// TIA Portal V18 program export: 1 tag tables, 0 data types, 5 data blocks, 11 code blocks (in call order from the OBs), 3 instance data blocks

VAR_GLOBAL   // PLC tag table "Default tag table"
   PB_MAIN_MOVE_R AT %I0.0 : Bool;
   PB_MAIN_MOVE_F AT %I0.1 : Bool;
   PB_MAIN_STOP AT %I0.2 : Bool;
   SENSOR_HOME AT %I0.3 : Bool;
   SENSOR_FINISH_1 AT %I0.4 : Bool;
   PB_EMERGENCY AT %I0.5 : Bool;
   PB_RESET AT %I0.6 : Bool;
   MAIN_COIL_R AT %Q0.0 : Bool;
   MAIN_COIL_F AT %Q0.1 : Bool;
   COIL_EMERGENCY AT %Q0.2 : Bool;
   System_Byte AT %MB1 : Byte;
   FirstScan AT %M1.0 : Bool;
   DiagStatusUpdate AT %M1.1 : Bool;
   AlwaysTRUE AT %M1.2 : Bool;
   AlwaysFALSE AT %M1.3 : Bool;
   Clock_Byte AT %MB0 : Byte;
   Clock_10Hz AT %M0.0 : Bool;
   Clock_5Hz AT %M0.1 : Bool;
   "Clock_2.5Hz" AT %M0.2 : Bool;
   Clock_2Hz AT %M0.3 : Bool;
   "Clock_1.25Hz" AT %M0.4 : Bool;
   Clock_1Hz AT %M0.5 : Bool;
   "Clock_0.625Hz" AT %M0.6 : Bool;
   "Clock_0.5Hz" AT %M0.7 : Bool;
   M1_RESET_COUNT AT %I0.7 : Bool;
   PB_M1_MOVE_R AT %I1.0 : Bool;
   PB_M1_MOVE_F AT %I1.1 : Bool;
   PB_M1_STOP AT %I1.2 : Bool;
   M1_COIL_R AT %Q0.3 : Bool;
   M1_COIL_F AT %Q0.4 : Bool;
   SENSOR_FINISH_2 AT %I1.3 : Bool;
   M2_RESET_COUNTER AT %I1.4 : Bool;
   PB_M2_MOVE_R AT %I1.5 : Bool;
   M2_COIL_R AT %Q0.5 : Bool;
   M2_COIL_F AT %Q0.6 : Bool;
   PB_M2_MOVE_F AT %I8.0 : Bool;
   PB_M2_STOP AT %I8.1 : Bool;
   DIVIDER_1 AT %Q8.0 : Bool;
   DIVIDER_2 AT %Q8.1 : Bool;
END_VAR

DATA_BLOCK "HMI_DB"   // DB20
{ S7_Optimized_Access := 'FALSE' }
VERSION : 0.1
// stored: AutoNumber true, DBAccessibleFromOPCUA true, IsOnlyStoredInLoadMemory false, IsWriteProtectedInAS false
   VAR
      MAIN_MOVE_F : Bool;
      MAIN_MOVE_R : Bool;
      MAIN_STOP : Bool;
      EMERGENCY : Bool;
      RESET : Bool;
      M1_MOVE_F : Bool;
      M1_MOVE_R : Bool;
      M1_STOP : Bool;
      RESET_COUNTER_1 : Bool;
      M2_MOVE_F : Bool;
      M2_MOVE_R : Bool;
      M2_STOP : Bool;
      RESET_COUNTER_2 : Bool;
      MAIN_FORWARD : Bool;
      MAIN_REVERSE : Bool;
      M1_FORWARD : Bool;
      M1_REVERSE : Bool;
      M2_FORWARD : Bool;
      M2_REVERSE : Bool;
   END_VAR
BEGIN
END_DATA_BLOCK

DATA_BLOCK "M1_I/O_DB"   // DB7
{ S7_Optimized_Access := 'FALSE' }
VERSION : 0.1
// stored: AutoNumber true, DBAccessibleFromOPCUA true, IsOnlyStoredInLoadMemory false, IsWriteProtectedInAS false
   VAR
      RESET_COUNTER : Bool;
      M1_MOVE_R : Bool;
      M1_MOVE_F : Bool;
      M1_STOP : Bool;
   END_VAR
BEGIN
END_DATA_BLOCK

DATA_BLOCK "M2_I/O_DB"   // DB19
{ S7_Optimized_Access := 'FALSE' }
VERSION : 0.1
// stored: AutoNumber true, DBAccessibleFromOPCUA true, IsOnlyStoredInLoadMemory false, IsWriteProtectedInAS false
   VAR
      RESET_COUNTER : Bool;
      M2_MOVE_R : Bool;
      M2_MOVE_F : Bool;
      M2_STOP : Bool;
   END_VAR
BEGIN
END_DATA_BLOCK

DATA_BLOCK "MAIN_I/O_DB"   // DB1
{ S7_Optimized_Access := 'FALSE' }
VERSION : 0.1
// stored: AutoNumber true, DBAccessibleFromOPCUA true, IsOnlyStoredInLoadMemory false, IsWriteProtectedInAS false
   VAR
      MAIN_MOVE_R : Bool;
      MAIN_MOVE_F : Bool;
      MAIN_STOP : Bool;
      SENSOR_HOME : Bool;
      SENSOR_FINISH_1 : Bool;
      SENSOR_FINISH_2 : Bool;
      EMERGENCY : Bool;
      RESET : Bool;
      MAIN_COIL_F : Bool;
      MAIN_COIL_R : Bool;
      COIL_EMERGENCY : Bool;
   END_VAR
BEGIN
END_DATA_BLOCK

DATA_BLOCK "STATES_DB"   // DB2
{ S7_Optimized_Access := 'FALSE' }
VERSION : 0.1
// stored: AutoNumber true, DBAccessibleFromOPCUA true, IsOnlyStoredInLoadMemory false, IsWriteProtectedInAS false
   VAR
      EMERGENCY_STATE : Bool;
      DIV_1 : Bool;
      DIV_2 : Bool;
      MAIN_WIND_DOWN : Bool;
      M1_WIND_DOWN : Bool;
      M2_WIND_DOWN : Bool;
      DIV1_COUNTING_READY : Bool;
      DIV2_COUNTING_READY : Bool;
   END_VAR
BEGIN
END_DATA_BLOCK

ORGANIZATION_BLOCK "Main"   // OB1, LAD, ProgramCycle
TITLE = "Main Program Sweep (Cycle)"
{ S7_Optimized_Access := 'TRUE' }
VERSION : 0.1
// stored: AutoNumber true, IsIECCheckEnabled false, SetENOAutomatically false
   VAR_INPUT
      Initial_Call : Bool;   // Initial call of this OB
      Remanence : Bool;   // =True, if remanent data are available
   END_VAR
BEGIN

REGION Network 1
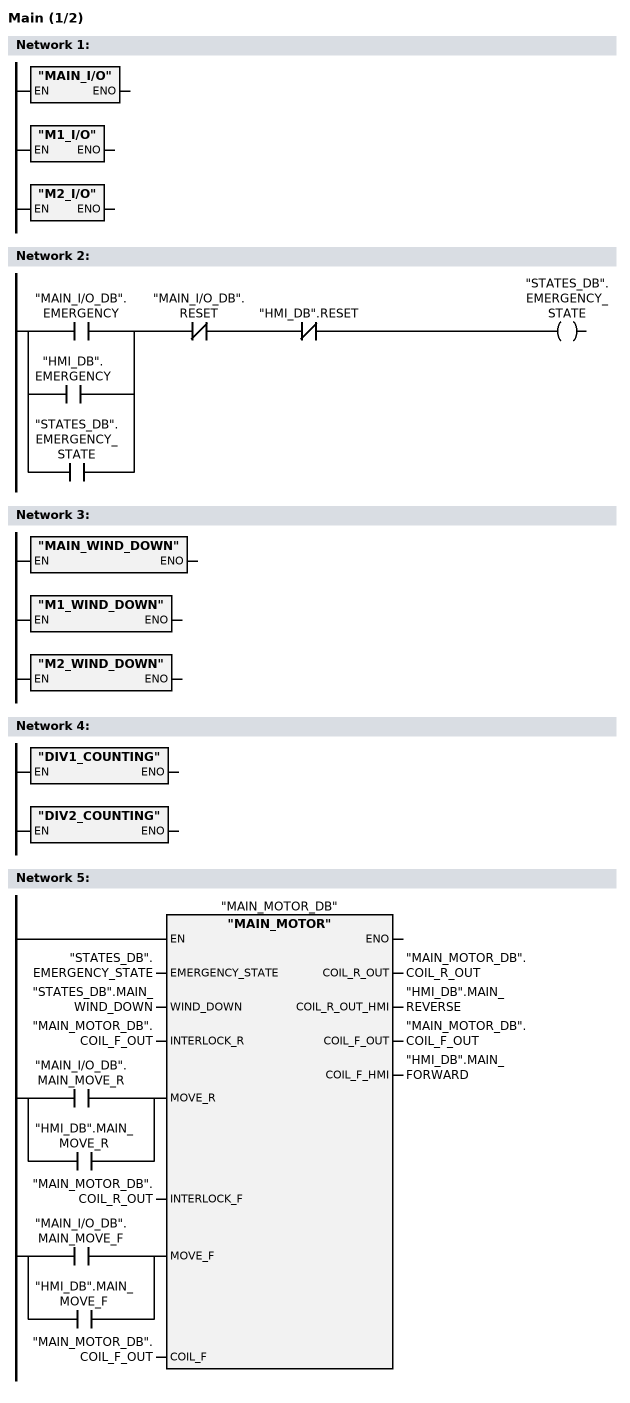
   RUNG wire#powerrail
      "MAIN_I/O"()
   END_RUNG
   RUNG wire#powerrail
      "M1_I/O"()
   END_RUNG
   RUNG wire#powerrail
      "M2_I/O"()
   END_RUNG
   // the same network as SCL:
   "MAIN_I/O"();
   "M1_I/O"();
   "M2_I/O"();
END_REGION

REGION Network 2
   RUNG wire#powerrail
      Contact( "MAIN_I/O_DB".EMERGENCY )
      wire#w1
      I_Contact( "MAIN_I/O_DB".RESET )
      I_Contact( "HMI_DB".RESET )
      Coil( "STATES_DB".EMERGENCY_STATE )
   END_RUNG
   RUNG wire#powerrail
      Contact( "HMI_DB".EMERGENCY )
   END_RUNG wire#w1
   RUNG wire#powerrail
      Contact( "STATES_DB".EMERGENCY_STATE )
   END_RUNG wire#w1
   // the same network as SCL:
   "STATES_DB".EMERGENCY_STATE := ("MAIN_I/O_DB".EMERGENCY OR "HMI_DB".EMERGENCY OR "STATES_DB".EMERGENCY_STATE) AND NOT "MAIN_I/O_DB".RESET AND NOT "HMI_DB".RESET;
END_REGION

REGION Network 3
   RUNG wire#powerrail
      "MAIN_WIND_DOWN"()
   END_RUNG
   RUNG wire#powerrail
      "M1_WIND_DOWN"()
   END_RUNG
   RUNG wire#powerrail
      "M2_WIND_DOWN"()
   END_RUNG
   // the same network as SCL:
   "MAIN_WIND_DOWN"();
   "M1_WIND_DOWN"();
   "M2_WIND_DOWN"();
END_REGION

REGION Network 4
   RUNG wire#powerrail
      "DIV1_COUNTING"()
   END_RUNG
   RUNG wire#powerrail
      "DIV2_COUNTING"()
   END_RUNG
   // the same network as SCL:
   "DIV1_COUNTING"();
   "DIV2_COUNTING"();
END_REGION

REGION Network 5
   RUNG wire#powerrail
      "MAIN_MOTOR_DB"(MOVE_R := wire#w1, MOVE_F := wire#w2, EMERGENCY_STATE := "STATES_DB".EMERGENCY_STATE, WIND_DOWN := "STATES_DB".MAIN_WIND_DOWN, INTERLOCK_R := "MAIN_MOTOR_DB".COIL_F_OUT, INTERLOCK_F := "MAIN_MOTOR_DB".COIL_R_OUT, COIL_F := "MAIN_MOTOR_DB".COIL_F_OUT, COIL_R_OUT => "MAIN_MOTOR_DB".COIL_R_OUT, COIL_R_OUT_HMI => "HMI_DB".MAIN_REVERSE, COIL_F_OUT => "MAIN_MOTOR_DB".COIL_F_OUT, COIL_F_HMI => "HMI_DB".MAIN_FORWARD)
   END_RUNG
   RUNG wire#powerrail
      Contact( "MAIN_I/O_DB".MAIN_MOVE_R )
   END_RUNG wire#w1
   RUNG wire#powerrail
      Contact( "HMI_DB".MAIN_MOVE_R )
   END_RUNG wire#w1
   RUNG wire#powerrail
      Contact( "MAIN_I/O_DB".MAIN_MOVE_F )
   END_RUNG wire#w2
   RUNG wire#powerrail
      Contact( "HMI_DB".MAIN_MOVE_F )
   END_RUNG wire#w2
   // the same network as SCL:
   "MAIN_MOTOR_DB"(EMERGENCY_STATE := "STATES_DB".EMERGENCY_STATE,   // "MAIN_MOTOR"
                   WIND_DOWN := "STATES_DB".MAIN_WIND_DOWN,
                   INTERLOCK_R := "MAIN_MOTOR_DB".COIL_F_OUT,
                   MOVE_R := "MAIN_I/O_DB".MAIN_MOVE_R OR "HMI_DB".MAIN_MOVE_R,
                   INTERLOCK_F := "MAIN_MOTOR_DB".COIL_R_OUT,
                   MOVE_F := "MAIN_I/O_DB".MAIN_MOVE_F OR "HMI_DB".MAIN_MOVE_F,
                   COIL_F := "MAIN_MOTOR_DB".COIL_F_OUT,
                   COIL_R_OUT => "MAIN_MOTOR_DB".COIL_R_OUT,
                   COIL_R_OUT_HMI => "HMI_DB".MAIN_REVERSE,
                   COIL_F_OUT => "MAIN_MOTOR_DB".COIL_F_OUT,
                   COIL_F_HMI => "HMI_DB".MAIN_FORWARD);
END_REGION

REGION Network 6
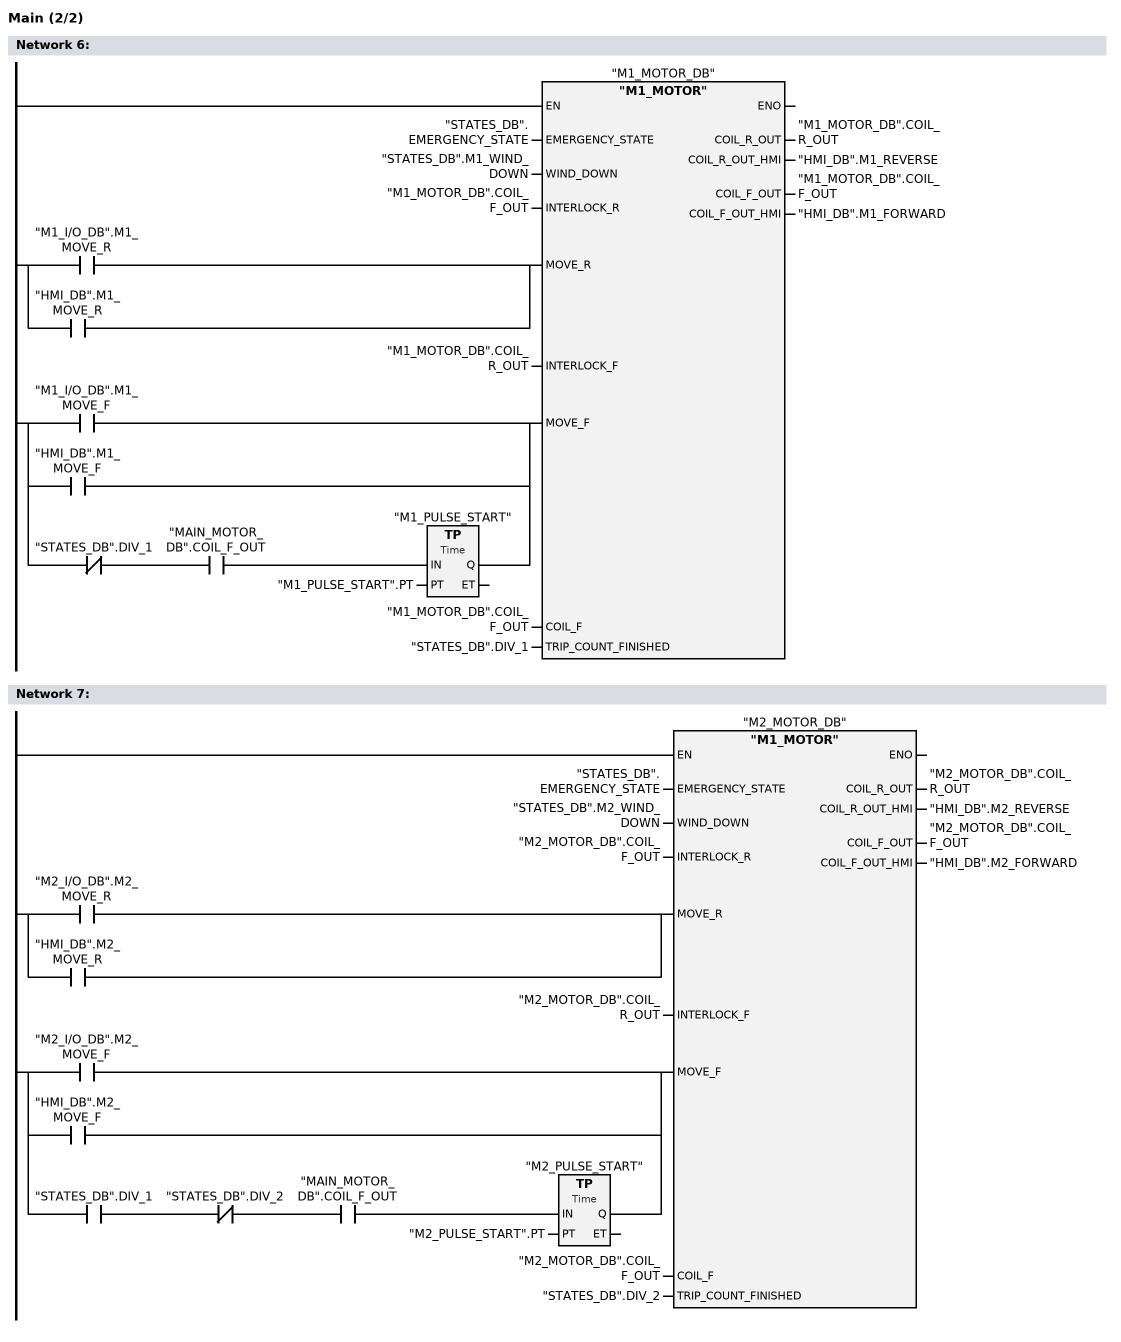
   RUNG wire#powerrail
      "M1_MOTOR_DB"(MOVE_R := wire#w1, MOVE_F := wire#w2, EMERGENCY_STATE := "STATES_DB".EMERGENCY_STATE, WIND_DOWN := "STATES_DB".M1_WIND_DOWN, INTERLOCK_R := "M1_MOTOR_DB".COIL_F_OUT, INTERLOCK_F := "M1_MOTOR_DB".COIL_R_OUT, COIL_F := "M1_MOTOR_DB".COIL_F_OUT, TRIP_COUNT_FINISHED := "STATES_DB".DIV_1, COIL_R_OUT => "M1_MOTOR_DB".COIL_R_OUT, COIL_R_OUT_HMI => "HMI_DB".M1_REVERSE, COIL_F_OUT => "M1_MOTOR_DB".COIL_F_OUT, COIL_F_OUT_HMI => "HMI_DB".M1_FORWARD)
   END_RUNG
   RUNG wire#powerrail
      Contact( "M1_I/O_DB".M1_MOVE_R )
   END_RUNG wire#w1
   RUNG wire#powerrail
      Contact( "HMI_DB".M1_MOVE_R )
   END_RUNG wire#w1
   RUNG wire#powerrail
      Contact( "M1_I/O_DB".M1_MOVE_F )
   END_RUNG wire#w2
   RUNG wire#powerrail
      Contact( "HMI_DB".M1_MOVE_F )
   END_RUNG wire#w2
   RUNG wire#powerrail
      I_Contact( "STATES_DB".DIV_1 )
      Contact( "MAIN_MOTOR_DB".COIL_F_OUT )
      { S7_Templates := "time_type := Time" } "M1_PULSE_START".TP(pt := "M1_PULSE_START".PT, et =>)
   END_RUNG wire#w2
   // the same network as SCL:
   "M1_PULSE_START".TP(IN := NOT "STATES_DB".DIV_1 AND "MAIN_MOTOR_DB".COIL_F_OUT, PT := "M1_PULSE_START".PT);
   "M1_MOTOR_DB"(EMERGENCY_STATE := "STATES_DB".EMERGENCY_STATE,   // "M1_MOTOR"
                 WIND_DOWN := "STATES_DB".M1_WIND_DOWN,
                 INTERLOCK_R := "M1_MOTOR_DB".COIL_F_OUT,
                 MOVE_R := "M1_I/O_DB".M1_MOVE_R OR "HMI_DB".M1_MOVE_R,
                 INTERLOCK_F := "M1_MOTOR_DB".COIL_R_OUT,
                 MOVE_F := "M1_I/O_DB".M1_MOVE_F OR "HMI_DB".M1_MOVE_F OR "M1_PULSE_START".Q,
                 COIL_F := "M1_MOTOR_DB".COIL_F_OUT,
                 TRIP_COUNT_FINISHED := "STATES_DB".DIV_1,
                 COIL_R_OUT => "M1_MOTOR_DB".COIL_R_OUT,
                 COIL_R_OUT_HMI => "HMI_DB".M1_REVERSE,
                 COIL_F_OUT => "M1_MOTOR_DB".COIL_F_OUT,
                 COIL_F_OUT_HMI => "HMI_DB".M1_FORWARD);
END_REGION

REGION Network 7
   RUNG wire#powerrail
      "M2_MOTOR_DB"(MOVE_R := wire#w1, MOVE_F := wire#w2, EMERGENCY_STATE := "STATES_DB".EMERGENCY_STATE, WIND_DOWN := "STATES_DB".M2_WIND_DOWN, INTERLOCK_R := "M2_MOTOR_DB".COIL_F_OUT, INTERLOCK_F := "M2_MOTOR_DB".COIL_R_OUT, COIL_F := "M2_MOTOR_DB".COIL_F_OUT, TRIP_COUNT_FINISHED := "STATES_DB".DIV_2, COIL_R_OUT => "M2_MOTOR_DB".COIL_R_OUT, COIL_R_OUT_HMI => "HMI_DB".M2_REVERSE, COIL_F_OUT => "M2_MOTOR_DB".COIL_F_OUT, COIL_F_OUT_HMI => "HMI_DB".M2_FORWARD)
   END_RUNG
   RUNG wire#powerrail
      Contact( "M2_I/O_DB".M2_MOVE_R )
   END_RUNG wire#w1
   RUNG wire#powerrail
      Contact( "HMI_DB".M2_MOVE_R )
   END_RUNG wire#w1
   RUNG wire#powerrail
      Contact( "M2_I/O_DB".M2_MOVE_F )
   END_RUNG wire#w2
   RUNG wire#powerrail
      Contact( "HMI_DB".M2_MOVE_F )
   END_RUNG wire#w2
   RUNG wire#powerrail
      Contact( "STATES_DB".DIV_1 )
      I_Contact( "STATES_DB".DIV_2 )
      Contact( "MAIN_MOTOR_DB".COIL_F_OUT )
      { S7_Templates := "time_type := Time" } "M2_PULSE_START".TP(pt := "M2_PULSE_START".PT, et =>)
   END_RUNG wire#w2
   // the same network as SCL:
   "M2_PULSE_START".TP(IN := "STATES_DB".DIV_1 AND NOT "STATES_DB".DIV_2 AND "MAIN_MOTOR_DB".COIL_F_OUT,
                       PT := "M2_PULSE_START".PT);
   "M2_MOTOR_DB"(EMERGENCY_STATE := "STATES_DB".EMERGENCY_STATE,   // "M1_MOTOR"
                 WIND_DOWN := "STATES_DB".M2_WIND_DOWN,
                 INTERLOCK_R := "M2_MOTOR_DB".COIL_F_OUT,
                 MOVE_R := "M2_I/O_DB".M2_MOVE_R OR "HMI_DB".M2_MOVE_R,
                 INTERLOCK_F := "M2_MOTOR_DB".COIL_R_OUT,
                 MOVE_F := "M2_I/O_DB".M2_MOVE_F OR "HMI_DB".M2_MOVE_F OR "M2_PULSE_START".Q,
                 COIL_F := "M2_MOTOR_DB".COIL_F_OUT,
                 TRIP_COUNT_FINISHED := "STATES_DB".DIV_2,
                 COIL_R_OUT => "M2_MOTOR_DB".COIL_R_OUT,
                 COIL_R_OUT_HMI => "HMI_DB".M2_REVERSE,
                 COIL_F_OUT => "M2_MOTOR_DB".COIL_F_OUT,
                 COIL_F_OUT_HMI => "HMI_DB".M2_FORWARD);
END_REGION
END_ORGANIZATION_BLOCK

FUNCTION "MAIN_I/O" : Void   // FC1, LAD
{ S7_Optimized_Access := 'TRUE' }
VERSION : 0.1
// stored: AutoNumber true, IsIECCheckEnabled false, SetENOAutomatically false, UDAEnableTagReadback false
BEGIN

REGION Network 1
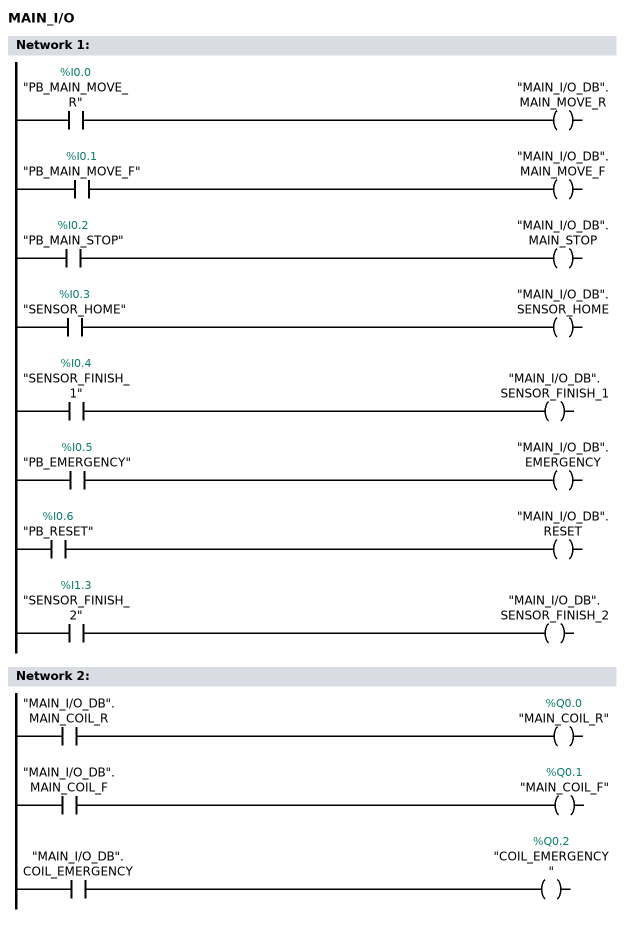
   RUNG wire#powerrail
      Contact( "PB_MAIN_MOVE_R" )
      Coil( "MAIN_I/O_DB".MAIN_MOVE_R )
   END_RUNG
   RUNG wire#powerrail
      Contact( "PB_MAIN_MOVE_F" )
      Coil( "MAIN_I/O_DB".MAIN_MOVE_F )
   END_RUNG
   RUNG wire#powerrail
      Contact( "PB_MAIN_STOP" )
      Coil( "MAIN_I/O_DB".MAIN_STOP )
   END_RUNG
   RUNG wire#powerrail
      Contact( "SENSOR_HOME" )
      Coil( "MAIN_I/O_DB".SENSOR_HOME )
   END_RUNG
   RUNG wire#powerrail
      Contact( "SENSOR_FINISH_1" )
      Coil( "MAIN_I/O_DB".SENSOR_FINISH_1 )
   END_RUNG
   RUNG wire#powerrail
      Contact( "PB_EMERGENCY" )
      Coil( "MAIN_I/O_DB".EMERGENCY )
   END_RUNG
   RUNG wire#powerrail
      Contact( "PB_RESET" )
      Coil( "MAIN_I/O_DB".RESET )
   END_RUNG
   RUNG wire#powerrail
      Contact( "SENSOR_FINISH_2" )
      Coil( "MAIN_I/O_DB".SENSOR_FINISH_2 )
   END_RUNG
   // the same network as SCL:
   "MAIN_I/O_DB".MAIN_MOVE_R := "PB_MAIN_MOVE_R";
   "MAIN_I/O_DB".MAIN_MOVE_F := "PB_MAIN_MOVE_F";
   "MAIN_I/O_DB".MAIN_STOP := "PB_MAIN_STOP";
   "MAIN_I/O_DB".SENSOR_HOME := "SENSOR_HOME";
   "MAIN_I/O_DB".SENSOR_FINISH_1 := "SENSOR_FINISH_1";
   "MAIN_I/O_DB".EMERGENCY := "PB_EMERGENCY";
   "MAIN_I/O_DB".RESET := "PB_RESET";
   "MAIN_I/O_DB".SENSOR_FINISH_2 := "SENSOR_FINISH_2";
END_REGION

REGION Network 2
   RUNG wire#powerrail
      Contact( "MAIN_I/O_DB".MAIN_COIL_R )
      Coil( "MAIN_COIL_R" )
   END_RUNG
   RUNG wire#powerrail
      Contact( "MAIN_I/O_DB".MAIN_COIL_F )
      Coil( "MAIN_COIL_F" )
   END_RUNG
   RUNG wire#powerrail
      Contact( "MAIN_I/O_DB".COIL_EMERGENCY )
      Coil( "COIL_EMERGENCY" )
   END_RUNG
   // the same network as SCL:
   "MAIN_COIL_R" := "MAIN_I/O_DB".MAIN_COIL_R;
   "MAIN_COIL_F" := "MAIN_I/O_DB".MAIN_COIL_F;
   "COIL_EMERGENCY" := "MAIN_I/O_DB".COIL_EMERGENCY;
END_REGION
END_FUNCTION

FUNCTION "M1_I/O" : Void   // FC4, LAD
{ S7_Optimized_Access := 'TRUE' }
VERSION : 0.1
// stored: AutoNumber true, IsIECCheckEnabled false, SetENOAutomatically false, UDAEnableTagReadback false
BEGIN

REGION Network 1
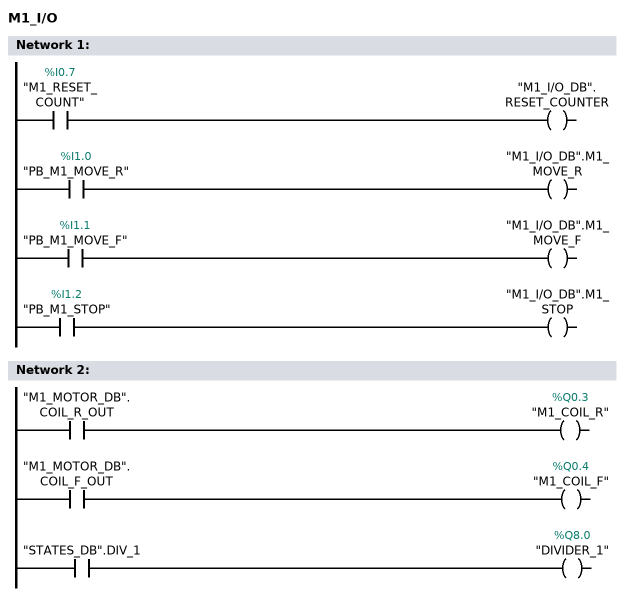
   RUNG wire#powerrail
      Contact( "M1_RESET_COUNT" )
      Coil( "M1_I/O_DB".RESET_COUNTER )
   END_RUNG
   RUNG wire#powerrail
      Contact( "PB_M1_MOVE_R" )
      Coil( "M1_I/O_DB".M1_MOVE_R )
   END_RUNG
   RUNG wire#powerrail
      Contact( "PB_M1_MOVE_F" )
      Coil( "M1_I/O_DB".M1_MOVE_F )
   END_RUNG
   RUNG wire#powerrail
      Contact( "PB_M1_STOP" )
      Coil( "M1_I/O_DB".M1_STOP )
   END_RUNG
   // the same network as SCL:
   "M1_I/O_DB".RESET_COUNTER := "M1_RESET_COUNT";
   "M1_I/O_DB".M1_MOVE_R := "PB_M1_MOVE_R";
   "M1_I/O_DB".M1_MOVE_F := "PB_M1_MOVE_F";
   "M1_I/O_DB".M1_STOP := "PB_M1_STOP";
END_REGION

REGION Network 2
   RUNG wire#powerrail
      Contact( "M1_MOTOR_DB".COIL_R_OUT )
      Coil( "M1_COIL_R" )
   END_RUNG
   RUNG wire#powerrail
      Contact( "M1_MOTOR_DB".COIL_F_OUT )
      Coil( "M1_COIL_F" )
   END_RUNG
   RUNG wire#powerrail
      Contact( "STATES_DB".DIV_1 )
      Coil( "DIVIDER_1" )
   END_RUNG
   // the same network as SCL:
   "M1_COIL_R" := "M1_MOTOR_DB".COIL_R_OUT;
   "M1_COIL_F" := "M1_MOTOR_DB".COIL_F_OUT;
   "DIVIDER_1" := "STATES_DB".DIV_1;
END_REGION
END_FUNCTION

FUNCTION "M2_I/O" : Void   // FC7, LAD
{ S7_Optimized_Access := 'TRUE' }
VERSION : 0.1
// stored: AutoNumber true, IsIECCheckEnabled false, SetENOAutomatically false, UDAEnableTagReadback false
BEGIN

REGION Network 1
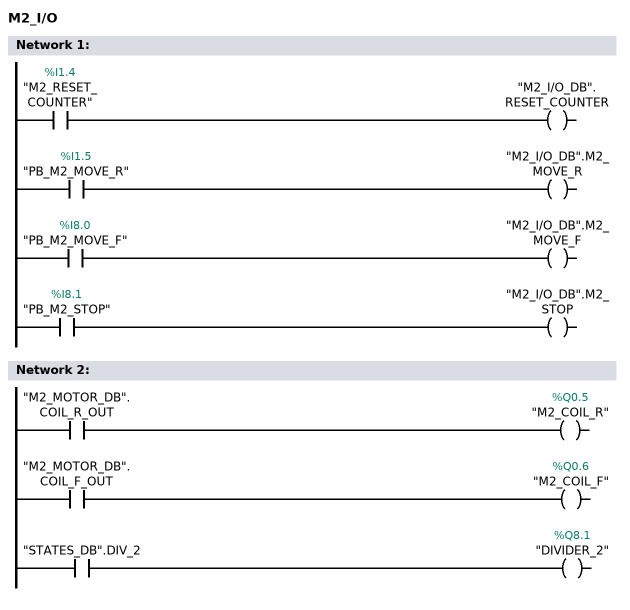
   RUNG wire#powerrail
      Contact( "M2_RESET_COUNTER" )
      Coil( "M2_I/O_DB".RESET_COUNTER )
   END_RUNG
   RUNG wire#powerrail
      Contact( "PB_M2_MOVE_R" )
      Coil( "M2_I/O_DB".M2_MOVE_R )
   END_RUNG
   RUNG wire#powerrail
      Contact( "PB_M2_MOVE_F" )
      Coil( "M2_I/O_DB".M2_MOVE_F )
   END_RUNG
   RUNG wire#powerrail
      Contact( "PB_M2_STOP" )
      Coil( "M2_I/O_DB".M2_STOP )
   END_RUNG
   // the same network as SCL:
   "M2_I/O_DB".RESET_COUNTER := "M2_RESET_COUNTER";
   "M2_I/O_DB".M2_MOVE_R := "PB_M2_MOVE_R";
   "M2_I/O_DB".M2_MOVE_F := "PB_M2_MOVE_F";
   "M2_I/O_DB".M2_STOP := "PB_M2_STOP";
END_REGION

REGION Network 2
   RUNG wire#powerrail
      Contact( "M2_MOTOR_DB".COIL_R_OUT )
      Coil( "M2_COIL_R" )
   END_RUNG
   RUNG wire#powerrail
      Contact( "M2_MOTOR_DB".COIL_F_OUT )
      Coil( "M2_COIL_F" )
   END_RUNG
   RUNG wire#powerrail
      Contact( "STATES_DB".DIV_2 )
      Coil( "DIVIDER_2" )
   END_RUNG
   // the same network as SCL:
   "M2_COIL_R" := "M2_MOTOR_DB".COIL_R_OUT;
   "M2_COIL_F" := "M2_MOTOR_DB".COIL_F_OUT;
   "DIVIDER_2" := "STATES_DB".DIV_2;
END_REGION
END_FUNCTION

FUNCTION "MAIN_WIND_DOWN" : Void   // FC2, LAD
{ S7_Optimized_Access := 'TRUE' }
VERSION : 0.1
// stored: AutoNumber true, IsIECCheckEnabled false, SetENOAutomatically false, UDAEnableTagReadback false
BEGIN

REGION Network 1
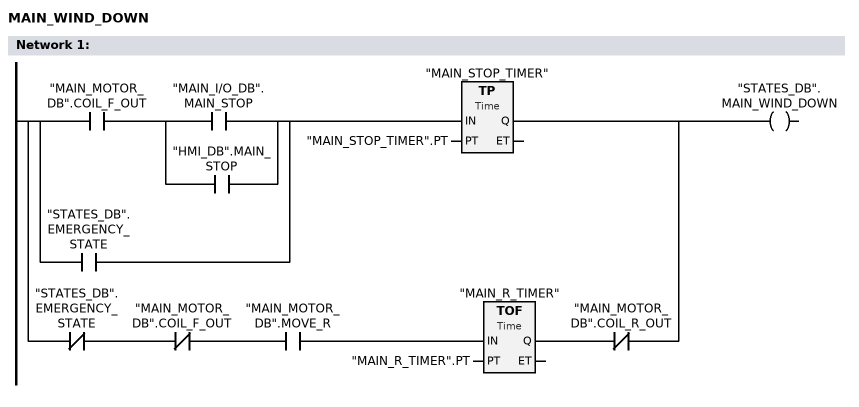
   RUNG wire#powerrail
      Contact( "MAIN_MOTOR_DB".COIL_F_OUT )
      wire#w1
      Contact( "MAIN_I/O_DB".MAIN_STOP )
      wire#w2
      { S7_Templates := "time_type := Time" } "MAIN_STOP_TIMER".TP(pt := "MAIN_STOP_TIMER".PT, et =>)
      wire#w3
      Coil( "STATES_DB".MAIN_WIND_DOWN )
   END_RUNG
   RUNG wire#w1
      Contact( "HMI_DB".MAIN_STOP )
   END_RUNG wire#w2
   RUNG wire#powerrail
      Contact( "STATES_DB".EMERGENCY_STATE )
   END_RUNG wire#w2
   RUNG wire#powerrail
      I_Contact( "STATES_DB".EMERGENCY_STATE )
      I_Contact( "MAIN_MOTOR_DB".COIL_F_OUT )
      Contact( "MAIN_MOTOR_DB".MOVE_R )
      { S7_Templates := "time_type := Time" } "MAIN_R_TIMER".TOF(pt := "MAIN_R_TIMER".PT, et =>)
      I_Contact( "MAIN_MOTOR_DB".COIL_R_OUT )
   END_RUNG wire#w3
   // the same network as SCL:
   "MAIN_STOP_TIMER".TP(IN := ("MAIN_MOTOR_DB".COIL_F_OUT AND ("MAIN_I/O_DB".MAIN_STOP OR "HMI_DB".MAIN_STOP)) OR "STATES_DB".EMERGENCY_STATE,
                        PT := "MAIN_STOP_TIMER".PT);
   "MAIN_R_TIMER".TOF(IN := NOT "STATES_DB".EMERGENCY_STATE AND NOT "MAIN_MOTOR_DB".COIL_F_OUT AND "MAIN_MOTOR_DB".MOVE_R,
                      PT := "MAIN_R_TIMER".PT);
   "STATES_DB".MAIN_WIND_DOWN := "MAIN_STOP_TIMER".Q OR ("MAIN_R_TIMER".Q AND NOT "MAIN_MOTOR_DB".COIL_R_OUT);
END_REGION
END_FUNCTION

FUNCTION "M1_WIND_DOWN" : Void   // FC5, LAD
{ S7_Optimized_Access := 'TRUE' }
VERSION : 0.1
// stored: AutoNumber true, IsIECCheckEnabled false, SetENOAutomatically false, UDAEnableTagReadback false
BEGIN

REGION Network 1
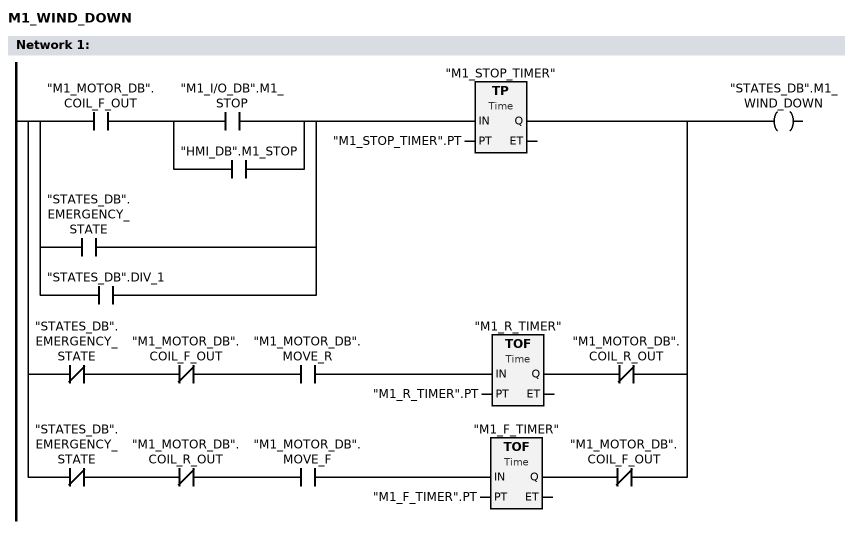
   RUNG wire#powerrail
      Contact( "M1_MOTOR_DB".COIL_F_OUT )
      wire#w1
      Contact( "M1_I/O_DB".M1_STOP )
      wire#w2
      { S7_Templates := "time_type := Time" } "M1_STOP_TIMER".TP(pt := "M1_STOP_TIMER".PT, et =>)
      wire#w3
      Coil( "STATES_DB".M1_WIND_DOWN )
   END_RUNG
   RUNG wire#w1
      Contact( "HMI_DB".M1_STOP )
   END_RUNG wire#w2
   RUNG wire#powerrail
      Contact( "STATES_DB".EMERGENCY_STATE )
   END_RUNG wire#w2
   RUNG wire#powerrail
      Contact( "STATES_DB".DIV_1 )
   END_RUNG wire#w2
   RUNG wire#powerrail
      I_Contact( "STATES_DB".EMERGENCY_STATE )
      I_Contact( "M1_MOTOR_DB".COIL_F_OUT )
      Contact( "M1_MOTOR_DB".MOVE_R )
      { S7_Templates := "time_type := Time" } "M1_R_TIMER".TOF(pt := "M1_R_TIMER".PT, et =>)
      I_Contact( "M1_MOTOR_DB".COIL_R_OUT )
   END_RUNG wire#w3
   RUNG wire#powerrail
      I_Contact( "STATES_DB".EMERGENCY_STATE )
      I_Contact( "M1_MOTOR_DB".COIL_R_OUT )
      Contact( "M1_MOTOR_DB".MOVE_F )
      { S7_Templates := "time_type := Time" } "M1_F_TIMER".TOF(pt := "M1_F_TIMER".PT, et =>)
      I_Contact( "M1_MOTOR_DB".COIL_F_OUT )
   END_RUNG wire#w3
   // the same network as SCL:
   "M1_STOP_TIMER".TP(IN := ("M1_MOTOR_DB".COIL_F_OUT AND ("M1_I/O_DB".M1_STOP OR "HMI_DB".M1_STOP)) OR "STATES_DB".EMERGENCY_STATE OR "STATES_DB".DIV_1,
                      PT := "M1_STOP_TIMER".PT);
   "M1_R_TIMER".TOF(IN := NOT "STATES_DB".EMERGENCY_STATE AND NOT "M1_MOTOR_DB".COIL_F_OUT AND "M1_MOTOR_DB".MOVE_R,
                    PT := "M1_R_TIMER".PT);
   "M1_F_TIMER".TOF(IN := NOT "STATES_DB".EMERGENCY_STATE AND NOT "M1_MOTOR_DB".COIL_R_OUT AND "M1_MOTOR_DB".MOVE_F,
                    PT := "M1_F_TIMER".PT);
   "STATES_DB".M1_WIND_DOWN := "M1_STOP_TIMER".Q OR ("M1_R_TIMER".Q AND NOT "M1_MOTOR_DB".COIL_R_OUT) OR ("M1_F_TIMER".Q AND NOT "M1_MOTOR_DB".COIL_F_OUT);
END_REGION
END_FUNCTION

FUNCTION "M2_WIND_DOWN" : Void   // FC8, LAD
{ S7_Optimized_Access := 'TRUE' }
VERSION : 0.1
// stored: AutoNumber true, IsIECCheckEnabled false, SetENOAutomatically false, UDAEnableTagReadback false
BEGIN

REGION Network 1
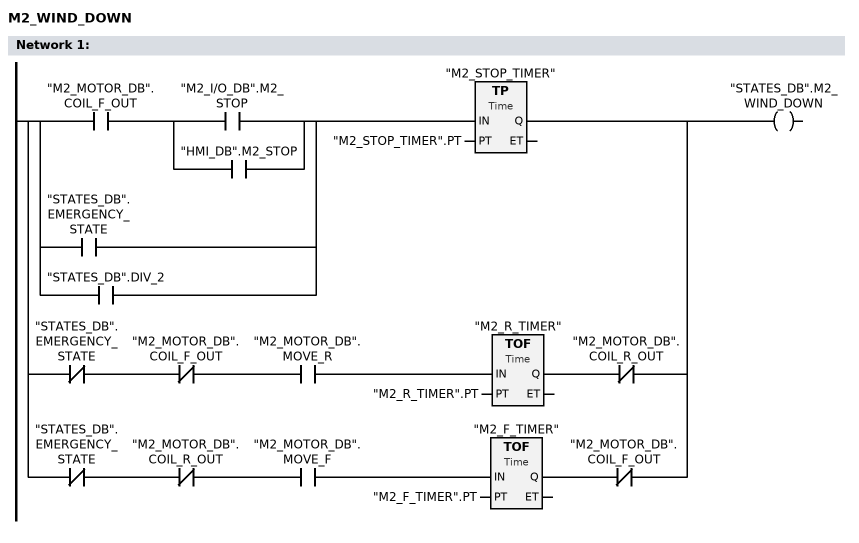
   RUNG wire#powerrail
      Contact( "M2_MOTOR_DB".COIL_F_OUT )
      wire#w1
      Contact( "M2_I/O_DB".M2_STOP )
      wire#w2
      { S7_Templates := "time_type := Time" } "M2_STOP_TIMER".TP(pt := "M2_STOP_TIMER".PT, et =>)
      wire#w3
      Coil( "STATES_DB".M2_WIND_DOWN )
   END_RUNG
   RUNG wire#w1
      Contact( "HMI_DB".M2_STOP )
   END_RUNG wire#w2
   RUNG wire#powerrail
      Contact( "STATES_DB".EMERGENCY_STATE )
   END_RUNG wire#w2
   RUNG wire#powerrail
      Contact( "STATES_DB".DIV_2 )
   END_RUNG wire#w2
   RUNG wire#powerrail
      I_Contact( "STATES_DB".EMERGENCY_STATE )
      I_Contact( "M2_MOTOR_DB".COIL_F_OUT )
      Contact( "M2_MOTOR_DB".MOVE_R )
      { S7_Templates := "time_type := Time" } "M2_R_TIMER".TOF(pt := "M2_R_TIMER".PT, et =>)
      I_Contact( "M2_MOTOR_DB".COIL_R_OUT )
   END_RUNG wire#w3
   RUNG wire#powerrail
      I_Contact( "STATES_DB".EMERGENCY_STATE )
      I_Contact( "M2_MOTOR_DB".COIL_R_OUT )
      Contact( "M2_MOTOR_DB".MOVE_F )
      { S7_Templates := "time_type := Time" } "M2_F_TIMER".TOF(pt := "M2_F_TIMER".PT, et =>)
      I_Contact( "M2_MOTOR_DB".COIL_F_OUT )
   END_RUNG wire#w3
   // the same network as SCL:
   "M2_STOP_TIMER".TP(IN := ("M2_MOTOR_DB".COIL_F_OUT AND ("M2_I/O_DB".M2_STOP OR "HMI_DB".M2_STOP)) OR "STATES_DB".EMERGENCY_STATE OR "STATES_DB".DIV_2,
                      PT := "M2_STOP_TIMER".PT);
   "M2_R_TIMER".TOF(IN := NOT "STATES_DB".EMERGENCY_STATE AND NOT "M2_MOTOR_DB".COIL_F_OUT AND "M2_MOTOR_DB".MOVE_R,
                    PT := "M2_R_TIMER".PT);
   "M2_F_TIMER".TOF(IN := NOT "STATES_DB".EMERGENCY_STATE AND NOT "M2_MOTOR_DB".COIL_R_OUT AND "M2_MOTOR_DB".MOVE_F,
                    PT := "M2_F_TIMER".PT);
   "STATES_DB".M2_WIND_DOWN := "M2_STOP_TIMER".Q OR ("M2_R_TIMER".Q AND NOT "M2_MOTOR_DB".COIL_R_OUT) OR ("M2_F_TIMER".Q AND NOT "M2_MOTOR_DB".COIL_F_OUT);
END_REGION
END_FUNCTION

FUNCTION "DIV1_COUNTING" : Void   // FC3, LAD
{ S7_Optimized_Access := 'TRUE' }
VERSION : 0.1
// stored: AutoNumber true, IsIECCheckEnabled false, SetENOAutomatically false, UDAEnableTagReadback false
BEGIN

REGION Network 1
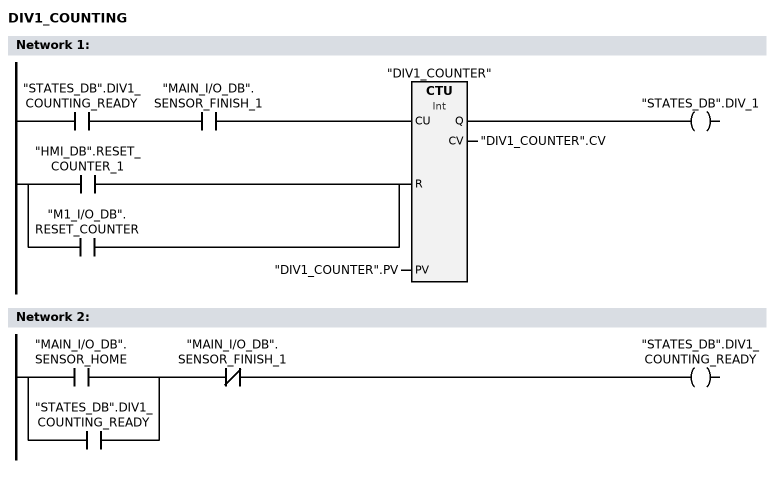
   RUNG wire#powerrail
      Contact( "STATES_DB".DIV1_COUNTING_READY )
      Contact( "MAIN_I/O_DB".SENSOR_FINISH_1 )
      { S7_Templates := "value_type := Int" } "DIV1_COUNTER".CTU(r := wire#w1, pv := "DIV1_COUNTER".PV, cv => "DIV1_COUNTER".CV)
      Coil( "STATES_DB".DIV_1 )
   END_RUNG
   RUNG wire#powerrail
      Contact( "HMI_DB".RESET_COUNTER_1 )
   END_RUNG wire#w1
   RUNG wire#powerrail
      Contact( "M1_I/O_DB".RESET_COUNTER )
   END_RUNG wire#w1
   // the same network as SCL:
   "DIV1_COUNTER".CTU(CU := "STATES_DB".DIV1_COUNTING_READY AND "MAIN_I/O_DB".SENSOR_FINISH_1,
                      R := "HMI_DB".RESET_COUNTER_1 OR "M1_I/O_DB".RESET_COUNTER,
                      PV := "DIV1_COUNTER".PV,
                      CV => "DIV1_COUNTER".CV);
   "STATES_DB".DIV_1 := "DIV1_COUNTER".Q;
END_REGION

REGION Network 2
   RUNG wire#powerrail
      Contact( "MAIN_I/O_DB".SENSOR_HOME )
      wire#w1
      I_Contact( "MAIN_I/O_DB".SENSOR_FINISH_1 )
      Coil( "STATES_DB".DIV1_COUNTING_READY )
   END_RUNG
   RUNG wire#powerrail
      Contact( "STATES_DB".DIV1_COUNTING_READY )
   END_RUNG wire#w1
   // the same network as SCL:
   "STATES_DB".DIV1_COUNTING_READY := ("MAIN_I/O_DB".SENSOR_HOME OR "STATES_DB".DIV1_COUNTING_READY) AND NOT "MAIN_I/O_DB".SENSOR_FINISH_1;
END_REGION
END_FUNCTION

FUNCTION "DIV2_COUNTING" : Void   // FC6, LAD
{ S7_Optimized_Access := 'TRUE' }
VERSION : 0.1
// stored: AutoNumber true, IsIECCheckEnabled false, SetENOAutomatically false, UDAEnableTagReadback false
BEGIN

REGION Network 1
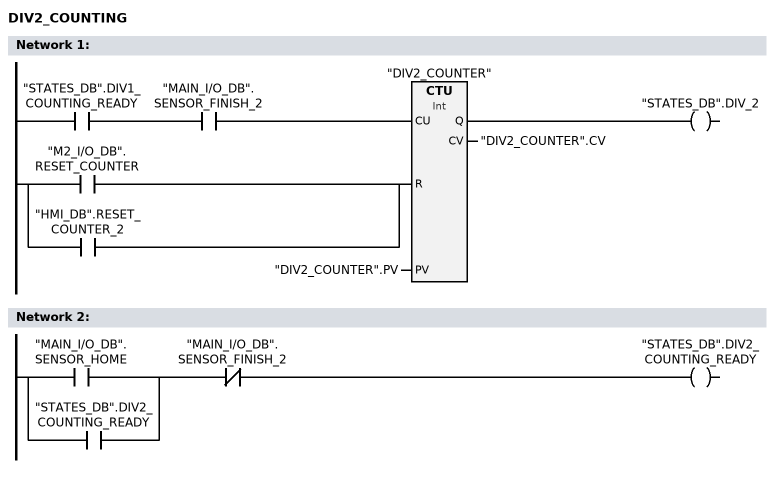
   RUNG wire#powerrail
      Contact( "STATES_DB".DIV1_COUNTING_READY )
      Contact( "MAIN_I/O_DB".SENSOR_FINISH_2 )
      { S7_Templates := "value_type := Int" } "DIV2_COUNTER".CTU(r := wire#w1, pv := "DIV2_COUNTER".PV, cv => "DIV2_COUNTER".CV)
      Coil( "STATES_DB".DIV_2 )
   END_RUNG
   RUNG wire#powerrail
      Contact( "M2_I/O_DB".RESET_COUNTER )
   END_RUNG wire#w1
   RUNG wire#powerrail
      Contact( "HMI_DB".RESET_COUNTER_2 )
   END_RUNG wire#w1
   // the same network as SCL:
   "DIV2_COUNTER".CTU(CU := "STATES_DB".DIV1_COUNTING_READY AND "MAIN_I/O_DB".SENSOR_FINISH_2,
                      R := "M2_I/O_DB".RESET_COUNTER OR "HMI_DB".RESET_COUNTER_2,
                      PV := "DIV2_COUNTER".PV,
                      CV => "DIV2_COUNTER".CV);
   "STATES_DB".DIV_2 := "DIV2_COUNTER".Q;
END_REGION

REGION Network 2
   RUNG wire#powerrail
      Contact( "MAIN_I/O_DB".SENSOR_HOME )
      wire#w1
      I_Contact( "MAIN_I/O_DB".SENSOR_FINISH_2 )
      Coil( "STATES_DB".DIV2_COUNTING_READY )
   END_RUNG
   RUNG wire#powerrail
      Contact( "STATES_DB".DIV2_COUNTING_READY )
   END_RUNG wire#w1
   // the same network as SCL:
   "STATES_DB".DIV2_COUNTING_READY := ("MAIN_I/O_DB".SENSOR_HOME OR "STATES_DB".DIV2_COUNTING_READY) AND NOT "MAIN_I/O_DB".SENSOR_FINISH_2;
END_REGION
END_FUNCTION

FUNCTION_BLOCK "MAIN_MOTOR"   // FB1, LAD
{ S7_Optimized_Access := 'TRUE' }
VERSION : 0.1
// stored: AutoNumber true, IsIECCheckEnabled false, IsRetainMemResEnabled false, MemoryReserve 100, SetENOAutomatically false, UDAEnableTagReadback false
   VAR_INPUT
      EMERGENCY_STATE : Bool;
      WIND_DOWN : Bool;
      INTERLOCK_R : Bool;
      MOVE_R : Bool;
      INTERLOCK_F : Bool;
      MOVE_F : Bool;
      COIL_F : Bool;
   END_VAR
   VAR_OUTPUT
      COIL_R_OUT : Bool;
      COIL_R_OUT_HMI : Bool;
      COIL_F_OUT : Bool;
      COIL_F_HMI : Bool;
   END_VAR
BEGIN

REGION Network 1
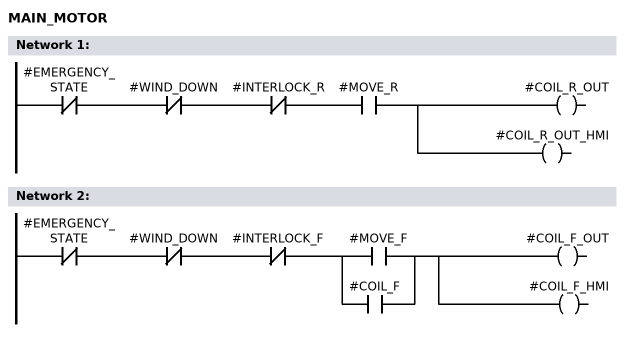
   RUNG wire#powerrail
      I_Contact( #EMERGENCY_STATE )
      I_Contact( #WIND_DOWN )
      I_Contact( #INTERLOCK_R )
      Contact( #MOVE_R )
      wire#w1
      Coil( #COIL_R_OUT )
   END_RUNG
   RUNG wire#w1
      Coil( #COIL_R_OUT_HMI )
   END_RUNG
   // the same network as SCL:
   #COIL_R_OUT := NOT #EMERGENCY_STATE AND NOT #WIND_DOWN AND NOT #INTERLOCK_R AND #MOVE_R;
   #COIL_R_OUT_HMI := #COIL_R_OUT;
END_REGION

REGION Network 2
   RUNG wire#powerrail
      I_Contact( #EMERGENCY_STATE )
      I_Contact( #WIND_DOWN )
      I_Contact( #INTERLOCK_F )
      wire#w1
      Contact( #MOVE_F )
      wire#w2
      Coil( #COIL_F_OUT )
   END_RUNG
   RUNG wire#w1
      Contact( #COIL_F )
   END_RUNG wire#w2
   RUNG wire#w2
      Coil( #COIL_F_HMI )
   END_RUNG
   // the same network as SCL:
   #COIL_F_OUT := NOT #EMERGENCY_STATE AND NOT #WIND_DOWN AND NOT #INTERLOCK_F AND (#MOVE_F OR #COIL_F);
   #COIL_F_HMI := #COIL_F_OUT;
END_REGION
END_FUNCTION_BLOCK

FUNCTION_BLOCK "M1_MOTOR"   // FB2, LAD
{ S7_Optimized_Access := 'TRUE' }
VERSION : 0.1
// stored: AutoNumber true, IsIECCheckEnabled false, IsRetainMemResEnabled false, MemoryReserve 100, SetENOAutomatically false, UDAEnableTagReadback false
   VAR_INPUT
      EMERGENCY_STATE : Bool;
      WIND_DOWN : Bool;
      INTERLOCK_R : Bool;
      MOVE_R : Bool;
      INTERLOCK_F : Bool;
      MOVE_F : Bool;
      COIL_F : Bool;
      TRIP_COUNT_FINISHED : Bool;
   END_VAR
   VAR_OUTPUT
      COIL_R_OUT : Bool;
      COIL_R_OUT_HMI : Bool;
      COIL_F_OUT : Bool;
      COIL_F_OUT_HMI : Bool;
   END_VAR
BEGIN

REGION Network 1
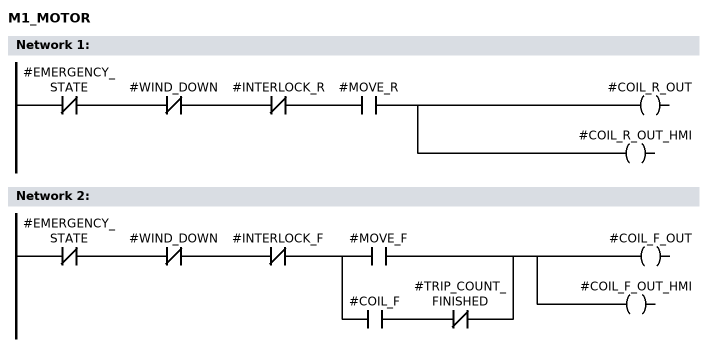
   RUNG wire#powerrail
      I_Contact( #EMERGENCY_STATE )
      I_Contact( #WIND_DOWN )
      I_Contact( #INTERLOCK_R )
      Contact( #MOVE_R )
      wire#w1
      Coil( #COIL_R_OUT )
   END_RUNG
   RUNG wire#w1
      Coil( #COIL_R_OUT_HMI )
   END_RUNG
   // the same network as SCL:
   #COIL_R_OUT := NOT #EMERGENCY_STATE AND NOT #WIND_DOWN AND NOT #INTERLOCK_R AND #MOVE_R;
   #COIL_R_OUT_HMI := #COIL_R_OUT;
END_REGION

REGION Network 2
   RUNG wire#powerrail
      I_Contact( #EMERGENCY_STATE )
      I_Contact( #WIND_DOWN )
      I_Contact( #INTERLOCK_F )
      wire#w1
      Contact( #MOVE_F )
      wire#w2
      Coil( #COIL_F_OUT )
   END_RUNG
   RUNG wire#w1
      Contact( #COIL_F )
      I_Contact( #TRIP_COUNT_FINISHED )
   END_RUNG wire#w2
   RUNG wire#w2
      Coil( #COIL_F_OUT_HMI )
   END_RUNG
   // the same network as SCL:
   #COIL_F_OUT := NOT #EMERGENCY_STATE AND NOT #WIND_DOWN AND NOT #INTERLOCK_F AND (#MOVE_F OR (#COIL_F AND NOT #TRIP_COUNT_FINISHED));
   #COIL_F_OUT_HMI := #COIL_F_OUT;
END_REGION
END_FUNCTION_BLOCK

DATA_BLOCK "M1_MOTOR_DB"   // DB8
VERSION : 0.1
// stored: AutoNumber true, DBAccessibleFromOPCUA true, InstanceOfName M1_MOTOR, InstanceOfType FB
"M1_MOTOR"
BEGIN
END_DATA_BLOCK

DATA_BLOCK "M2_MOTOR_DB"   // DB13
VERSION : 0.1
// stored: AutoNumber true, DBAccessibleFromOPCUA true, InstanceOfName M1_MOTOR, InstanceOfType FB
"M1_MOTOR"
BEGIN
END_DATA_BLOCK

DATA_BLOCK "MAIN_MOTOR_DB"   // DB3
VERSION : 0.1
// stored: AutoNumber true, DBAccessibleFromOPCUA true, InstanceOfName MAIN_MOTOR, InstanceOfType FB
"MAIN_MOTOR"
BEGIN
END_DATA_BLOCK
